Fanuc KAREL source: kt00448.KL

-- PROVISIONAL review KL for V1013-1; original PC SHA256 ad9906ff42a1b1857146be5f3b0ed485ce67cd43a55ff7f6e87474c08b48400b
-- Incomplete behavior may be omitted. Consult companion uncertainty JSON. Do not deploy.
PROGRAM KT00448
%NOLOCKGROUP
VAR
  R2 : REAL
  OUT : BOOLEAN
-- UNRESOLVED_DECL Y1 type=002018
BEGIN
  -- UNRESOLVED_PC offsets 5-19; opcodes 2E,22,9D,33,B2
  -- UNRESOLVED_PC offsets 24-35; opcodes 2E,23
  -- UNRESOLVED_PC offsets 40-65; opcodes 22,9D,33,B1,21,29,64,29,72,23
  -- UNRESOLVED_PC offsets 70-74; opcodes 7F
END KT00448
